FUNCTION_BLOCK STATION_CONTROL
  {SET_ATTRIBUTE(OpcUa, SERVICE)}
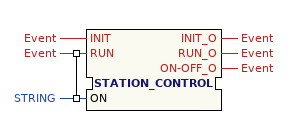
  EVENT_INPUT
    INIT;
    RUN WITH ON; {SET_ATTRIBUTE(OpcUa, Method)}
  END_EVENT
  EVENT_OUTPUT
    INIT_O;
    RUN_O;
    ON-OFF_O;
  END_EVENT
  VAR_INPUT
    ON : STRING;
  END_VAR
END_FUNCTION_BLOCK
